# EPICS substitutions: viocs/si_ps/si_psApp/Db/sdp1.substitutions
file "db/individual.db" {
    pattern { family, pos, num }
        { "SDP1", "02C4", "" }
        { "SDP1", "03C1", "" }
        { "SDP1", "06C4", "" }
        { "SDP1", "07C1", "" }
        { "SDP1", "12C4", "" }
        { "SDP1", "11C1", "" }
        { "SDP1", "14C4", "" }
        { "SDP1", "15C1", "" }
        { "SDP1", "18C4", "" }
        { "SDP1", "19C1", "" }
}
